{attribute 'qualified_only'}
{attribute 'strict'}
TYPE nUnderPressureTestErrorCodes :
(
	TestTimeOut := 860,
	SafetyError := 861
	
);
END_TYPE

(* stored: Version 1.1.0.1, ProductVersion 3.1.4024.13
   DUT nUnderPressureTestErrorCodes: Id {839be7ad-47d7-4b5b-be1c-cff2c2d26016} *)
